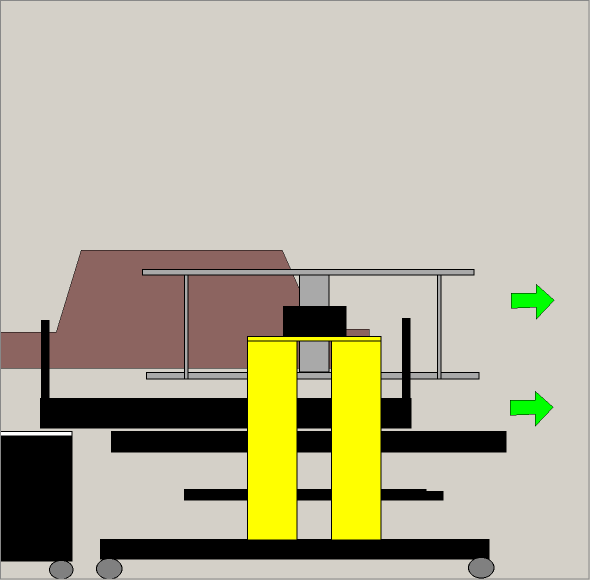
VISUALIZATION unloadSpaScreen  // 590x580
    Polygon (-12,368) (-11,332) (56,332) (81,250) (282,250) (317,329) (369,329) (369,367) (369,368)
    Rectangle (40,398 371x30)
    Rectangle (265,308 98x30), angle 90
    Rectangle (146,372 333x7)
    Rectangle (184,489 242x11), angle 25
    Rectangle (200,491 243x9), angle 336
    Rectangle (111,431 395x21)
    Rectangle (100,539 389x20)
    Rectangle (247,340 50x200)
    Rectangle (331,340 50x200)
    Ellipse (468,557 26x21)
    Ellipse (96,558 26x21)
    Rectangle (247,336 134x5)
    Rectangle (437,274 4x105)
    Rectangle (184,274 4x105)
    Rectangle (142,269 332x6)
    Rectangle (283,306 63x30)
    Rectangle (402,318 8x101)
    Rectangle (41,320 8x101)
    Polygon (511,303) (511,308) (536,307) (536,319) (554,300) (536,284) (536,293) (511,293)
    Polygon (510,410) (510,415) (535,414) (535,426) (553,407) (535,391) (535,400) (510,400)
    Rectangle (0,431 72x5)
    Rectangle (0,436 72x125)
    Ellipse (49,560 24x19)
END_VISUALIZATION

(* stored: Version 1.1.0.1, ProductVersion 3.1.4024.13
   Visu unloadSpaScreen: Id {e65d13bc-82ad-4f56-a491-fa4aaf0fe437} *)
